FUNCTION_BLOCK SS5a_AirNozzle (* Basic FB with empty ECC *)
  (* Standard: 61499-2 *)
  (* Version 1.0, 2024-10-03, DEVIASH *)
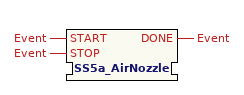
  EVENT_INPUT
    START;
    STOP;
  END_EVENT
  EVENT_OUTPUT
    DONE;
  END_EVENT
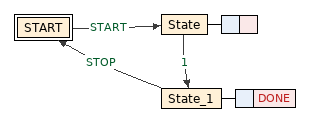
  EC_STATES
    START; (* Initial State *)
    State;
    State_1 : -> DONE;
  END_STATES
  EC_TRANSITIONS
    START TO State := START;
    State_1 TO START := STOP;
    State TO State_1 := 1;
  END_TRANSITIONS
END_FUNCTION_BLOCK
